FUNCTION_BLOCK NCITable
VAR_INPUT
END_VAR
VAR_OUTPUT
END_VAR
VAR
	nciTable : ST_NciFeedGroupTable;
END_VAR

;

END_FUNCTION_BLOCK

(* stored: Version 1.1.0.1, ProductVersion 3.1.4020.3
   POU NCITable: Id {39df6223-76ff-44a1-bd5a-f99611d1d1ef}, SpecialFunc None *)
